TYPE udtHourlyData :
STRUCT
	GoodCount :DINT :=0;
	ScrapCount :DINT :=0;	
END_STRUCT
END_TYPE

(* stored: Version 1.1.0.1, ProductVersion 3.1.4020.6
   DUT udtHourlyData: Id {b9ba998e-1b9a-478b-bdd0-cb05a6b759bb} *)
